// TIA Portal V18 export
// export: Created 2026-03-12T16:04:34.4454008Z, ExportSetting WithDefaults, DisplayName Totally Integrated Automation Portal, DisplayVersion V18 Update 5, DisplayName TIA Portal Openness, DisplayVersion V18 Update 5, DisplayName TIA Portal Version Control Interface, DisplayVersion V18, DisplayName SINAMICS Startdrive Advanced, DisplayVersion V18, DisplayName SINAMICS Startdrive G130, G150, S120, S150, SINAMICS MV, S210, DisplayVersion V18, DisplayName SINAMICS Startdrive G110M, G120, G120C, G120D, G120P, G115D, DisplayVersion V18, DisplayName STEP 7 Professional, DisplayVersion V18 Update 5, DisplayName STEP 7 Safety, DisplayVersion V18, DisplayName WinCC Professional, DisplayVersion V18 Update 5
FUNCTION_BLOCK "FB AFERIÇÃO INVERSORES"   // FB2, LAD
{ S7_Optimized_Access := 'TRUE' }
VERSION : 0.1
// Os sinais de campo são recebidos em corrente (4-20mA) e representados pelo fundo de escala do CLP. Este bloco faz a conversão do sinal para a leitura real da medição.
// 
// Network 1: Ajuste do fundo de escala aos parâmetros de aferição
// Network 2: Cálculo da equação da reta para definir a leitura atual da entrada analógica
// Network 3: Setando o alarme SEM 4mA na entrada digital caso seja rompida
// stored: AutoNumber true, IsIECCheckEnabled false, IsRetainMemResEnabled false, MemoryReserve 100, SetENOAutomatically false, UDAEnableTagReadback false
   VAR_INPUT
      ANALOG_IN_4a20mA : Int;   // Entrada do sinal analógico
      Y1_CONFIG : Int;   // Fundo de escala mínimo para o CLP
      Y2_CONFIG : Int;   // Fundo de escala máximo para o CLP
      X1_CONFIG : Int;   // Fundo de escala mínimo para o equipamento
      X2_CONFIG : Int;   // Fundo de escala máximo para o equipamento
      COMANDO : Int;   // Comando enviado da IHM/SCADA para aferir determinado equipamento
      COMANDO_VALOR : Int;   // Valor comparativo para executar o Bloco FB
      GRANDEZA_MAX : Int;   // Referência a grandeza maxima no qual o bloco vai utilizar para fazer a curva da reta
   END_VAR
   VAR_OUTPUT
      ANALOG_OUT_4a20mA : Real;   // Saída do sinal analógico já aferido
      ALARME_SEM_4mA : Bool;   // 1 = Entrada sem 4mA, indicando erro; 0 = Entrada OK
      RANGE_MIN_CADASTRADO : Int;   // Valor do cadastro máximo armazenado para visualizar na IHM
      RANGE_MAX_CADASTRADO : Int;   // Valor do cadastro mínimo armazenado para visualizar na IHM
   END_VAR
   VAR
      ANALOG_IN_LIMITED : Int;   // Tratamento de erro do sinal analógico para capturar apenas leituras que estão dentro do range do CLP
      ANALOG_IN_LIMITED_REAL : UInt;   // Saída do sinal ajustado conforme a grandeza máxima
      STATIC_X1 : UInt;   // Fundo de escala mínimo para o equipamento (Instanciado no FB)
      STATIC_X2 : UInt;   // Fundo de escala máximo para o equipamento (Instanciado no FB)
      STATIC_Y1 : UInt;   // Fundo de escala mínimo para o CLP (Instanciado no FB)
      STATIC_Y2 : UInt;   // Fundo de escala máximo para o CLP (Instanciado no FB)
      STATIC_GRANDEZA_MAX : UInt;   // Grandeza máxima do equipamento
      AJUSTAR_CURVA : Bool;   // Memória para mover as entradas às instâncias
      PONTO_ZERO : Int;   // Range mínimo do equipamento quando é diferente de 0
      ALARME_RESET : TOF_TIME;   // Reset do alarme Sem 4mA ao estabilizar o sinal
      PULSO_AJUSTAR : Bool;   // Pulso para realizar a aferição da curva
   END_VAR
   VAR_TEMP   // added for the SCL form of the ladder/FBD networks
      _w1 : Bool;
   END_VAR
BEGIN

REGION Network 1: Ajuste do fundo de escala aos parâmetros de aferição
   // X1_CONFIG = Fundo de escala mínimo para o equipamento
   // X2_CONFIG = Fundo de escala máximo para o equipamento
   // Y1_CONFIG = Fundo de escala mínimo para o CLP
   // Y2_CONFIG = Fundo de escala máximo para o CLP
   // GRANDEZA_MAX = Referência a grandeza maxima no qual o bloco vai utilizar para fazer a curva da reta
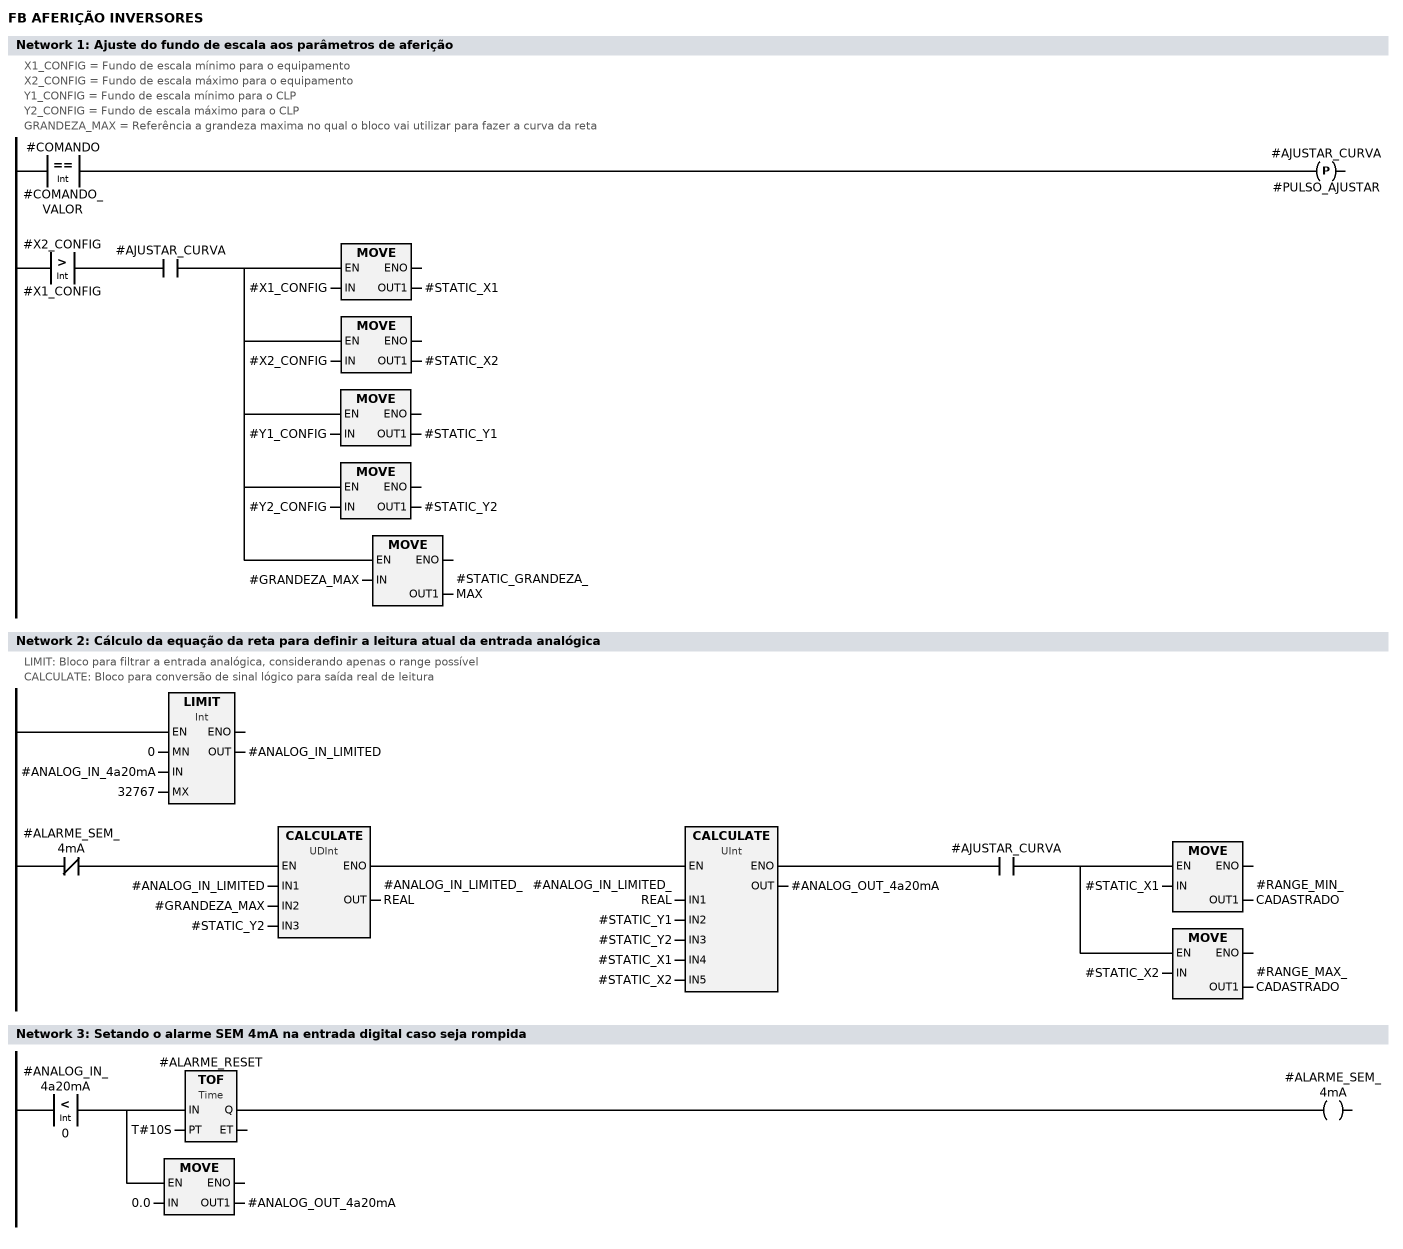
   #_w1 := #COMANDO = #COMANDO_VALOR;
   #AJUSTAR_CURVA := #_w1 AND NOT #PULSO_AJUSTAR;   // rising edge
   #PULSO_AJUSTAR := #_w1;
   IF (#X2_CONFIG > #X1_CONFIG) AND #AJUSTAR_CURVA THEN
       #STATIC_X1 := #X1_CONFIG;
       #STATIC_X2 := #X2_CONFIG;
       #STATIC_Y1 := #Y1_CONFIG;
       #STATIC_Y2 := #Y2_CONFIG;
       #STATIC_GRANDEZA_MAX := #GRANDEZA_MAX;
   END_IF;
END_REGION

REGION Network 2: Cálculo da equação da reta para definir a leitura atual da entrada analógica
   // LIMIT: Bloco para filtrar a entrada analógica, considerando apenas o range possível
   // CALCULATE: Bloco para conversão de sinal lógico para saída real de leitura
   RUNG wire#powerrail
      { S7_Templates := "value_type := Int" } Limit(mn := 0, in := #ANALOG_IN_4a20mA, mx := 32767, out => #ANALOG_IN_LIMITED)
   END_RUNG
   RUNG wire#powerrail
      I_Contact( #ALARME_SEM_4mA )
      { S7_Templates := "SrcType := UDInt"; S7_Expression := "IN1 * IN3 / IN2" } Calculate(in1 := #ANALOG_IN_LIMITED, in2 := #GRANDEZA_MAX, in3 := #STATIC_Y2, out => #ANALOG_IN_LIMITED_REAL)
      { S7_Templates := "SrcType := UInt"; S7_Expression := "(IN1 - IN2) * (IN5 - IN4) / (IN3 - IN2)" } Calculate(in1 := #ANALOG_IN_LIMITED_REAL, in2 := #STATIC_Y1, in3 := #STATIC_Y2, in4 := #STATIC_X1, in5 := #STATIC_X2, out => #ANALOG_OUT_4a20mA)
      Contact( #AJUSTAR_CURVA )
      wire#w1
      Move(in := #STATIC_X1, out1 => #RANGE_MIN_CADASTRADO)
   END_RUNG
   RUNG wire#w1
      Move(in := #STATIC_X2, out1 => #RANGE_MAX_CADASTRADO)
   END_RUNG
   // the same network as SCL:
   #ANALOG_IN_LIMITED := LIMIT(MN := 0, IN := #ANALOG_IN_4a20mA, MX := 32767);
   IF NOT #ALARME_SEM_4mA THEN
       #ANALOG_IN_LIMITED_REAL := #ANALOG_IN_LIMITED * #STATIC_Y2 / #GRANDEZA_MAX;
       #ANALOG_OUT_4a20mA := (#ANALOG_IN_LIMITED_REAL - #STATIC_Y1) * (#STATIC_X2 - #STATIC_X1) / (#STATIC_Y2 - #STATIC_Y1);
   END_IF;
   IF NOT #ALARME_SEM_4mA AND #AJUSTAR_CURVA THEN
       #RANGE_MIN_CADASTRADO := #STATIC_X1;
       #RANGE_MAX_CADASTRADO := #STATIC_X2;
   END_IF;
END_REGION

REGION Network 3: Setando o alarme SEM 4mA na entrada digital caso seja rompida
   RUNG wire#powerrail
      { S7_Templates := "SrcType := Int" } LT_Contact(in1 := #ANALOG_IN_4a20mA, in2 := 0)
      wire#w1
      { S7_Templates := "time_type := Time" } #ALARME_RESET.TOF(pt := T#10S, et =>)
      Coil( #ALARME_SEM_4mA )
   END_RUNG
   RUNG wire#w1
      Move(in := 0.0, out1 => #ANALOG_OUT_4a20mA)
   END_RUNG
   // the same network as SCL:
   #_w1 := #ANALOG_IN_4a20mA < 0;
   #ALARME_RESET(IN := #_w1, PT := T#10S);   // TOF
   #ALARME_SEM_4mA := #ALARME_RESET.Q;
   IF #_w1 THEN #ANALOG_OUT_4a20mA := 0.0; END_IF;
END_REGION
END_FUNCTION_BLOCK
